// SIMATIC S7-200 project (STEP 7-Micro/WIN), CPU 226 REL 01.00

SYMBOL_TABLE SYM1
命令               VB100
bcc              VB101
bcc_ath          VB102
bcc_0            VB103
地址半高             VB104
地址半低             VB105
返回BCC            VB106
地址               VD110
位数h              VB114
位数               VB115
接收缓冲开始           VB120
接收缓冲结束           VB148
发送缓冲开始           VB149
发送缓冲结束           VB190
接受错缓冲开始          VB191
接受错缓冲结束          VB194
写到plc正确缓冲开始      VB195
写到plc正确缓冲结束      VB198
END_SYMBOL_TABLE

ORGANIZATION_BLOCK MAIN:OB1
TITLE=【101】环保处理厂的焚烧炉PLC控制程序
// 系统通过PLC管理焚烧炉的启动、运行、停止和故障处理，支持多设备协同工作。
// 操作员通过置位系统启动标志启动系统，随后系统根据1#燃烧室温度传感器和2#燃烧室温度传感器的反馈自动运行。焚烧过程由1#燃烧室燃烧器控制、2#燃烧室1#燃烧器控制和2#燃烧室2#燃烧器控制负责，但1#燃烧室燃烧器控制只能在2#燃烧室1#燃烧器控制未运行时启动，同样2#燃烧室1#燃烧器控制只能在1#燃烧室燃烧器控制未运行时启动，以防止焚烧炉过热或设备损坏。废液通过酸性废液输送泵控制和碱性废液输送泵控制输送，其中酸性废液输送泵控制和碱性废液输送泵控制交替运行，确保废液分开输送。接着，酸性废液喷嘴控制、碱性废液喷嘴控制和502废液喷嘴控制负责将废液喷射到焚烧炉内，且酸性废液喷嘴控制在废液输送时打开，确保废液均匀分布。
// 炉内气流由引风机控制和鼓风机控制维持，两者协同运行，保证氧气供应和废气排放顺畅。焚烧后的废渣由出渣机控制排出，且出渣机控制在焚烧结束后启动，避免堵塞。废气处理依赖药剂输送泵1控制至药剂输送泵4控制输送中和剂，其中药剂输送泵1控制在药剂可用时运行，防止泵空转；药剂池搅拌机控制确保药剂均匀。随后，能量回收通过余热锅炉1#给水泵控制和余热锅炉2#给水泵控制实现，余热锅炉1#给水泵控制在需要补水时启动，避免锅炉过压。
// 废气进一步通过喷淋塔电动阀控制和石灰池电磁阀控制处理，其中喷淋塔电动阀控制根据废气温度调整，确保处理效果。1#冷却塔风扇控制和2#冷却塔风扇控制冷却循环水，软水冷却泵控制辅助冷却。系统配备故障检测，如超温、熄火等，异常时通过故障报警灯控制提示操作员。停止时，系统启动标志复位，所有设备（如1#燃烧室燃烧器控制等）随之复位，确保安全关闭。
BEGIN
Network 1
LD     SM0.1
MOVB   16#9, SMB30           //口1波特率9600,N,8,1
ATCH   INT_0:INT0, 8         //口1中断,中断程序0
MOVW   16#3032, VW104        //PLC地址(01)0-30,1-31
MOVD   16#3030705, VD191     //VB191=3,VB192=3,7,5
R      M0.0, 8               //初始化MB0
MOVD   16#3030605, VD195     //接收错缓冲区
ENI
Network 2
LD     SM0.7
=      SM30.0
?000
Network 3
LD     M0.3                  //接收正确
O      M0.4                  //接收错
CALL   SBR_0:SBR0            //答复计算机
Network 4 // 子程序调用
// 
// 
LD     SM0.0
CALL   SBR_1:SBR1
CALL   SBR_2:SBR2
CALL   SBR_3:SBR3
CALL   SBR_4:SBR4
Network 5 // 系统启动
// 
// 
LD     M6.6
=      M10.0
Network 6
LD     SM0.0
MOVR   VD208, VD600
-R     5.0, VD600
MOVR   VD212, VD604
-R     5.0, VD604
MOVR   VD228, VD608
-R     5.0, VD608
MOVR   VD236, VD612
-R     5.0, VD612
MOVR   VD224, VD616
-R     5.0, VD616
MOVR   VD232, VD620
-R     5.0, VD620
Network 7 // 系统启动   1#燃烧室燃烧器控制
//  
// NETWORK COMMENTS
//  
// 
LD     SM0.0
A      M10.0
LPS
A      M6.5
LPS
S      Q4.1, 1
AR<    VD1216, VD600
S      Q4.2, 1
LRD
AR<    VD1216, VD604
S      Q4.3, 1
LRD
AR>    VD1216, VD208
R      Q4.2, 2
LRD
AR>    VD1216, VD212
R      Q4.3, 1
LPP
A      M14.1
R      Q4.2, 2
LPP
AN     M6.5
R      Q4.1, 3
Network 8 // 2#燃烧室1#燃烧器控制
//  
// NETWORK COMMENTS
//  
// 
LD     SM0.0
A      M10.0
LPS
A      M11.1
LPS
S      Q4.4, 1
AR<    VD1416, VD608
S      Q4.6, 1
LRD
AR<    VD1416, VD612
S      Q4.5, 1
LRD
AR>    VD1416, VD228
R      Q4.6, 1
LRD
AR>    VD1416, VD236
R      Q4.5, 1
LPP
A      M14.2
R      Q4.5, 2
LPP
AN     M11.1
R      Q4.4, 3
Network 9 // 2#燃烧室2#燃烧器控制
//  
// NETWORK COMMENTS
//  
// 
LD     SM0.0
A      M10.0
LPS
A      M11.3
LPS
S      Q4.7, 1
AR<    VD1416, VD616
S      Q5.1, 1
LRD
AR<    VD1416, VD620
S      Q5.0, 1
LRD
AR>    VD1416, VD224
R      Q5.1, 1
LRD
AR>    VD1416, VD232
R      Q5.0, 1
LPP
A      M14.3
R      Q5.0, 2
LPP
AN     M11.3
R      Q4.7, 3
Network 10 // 酸性废液输送泵控制
// 
// 
LD     SM0.0
LPS
A      M10.0
A      M10.2
S      Q2.3, 1
LPP
AN     M10.2
R      Q2.3, 1
Network 11 // 碱性废液输送泵控制
// 
// 
LD     SM0.0
LPS
A      M10.0
A      M10.4
S      Q2.4, 1
LPP
AN     M10.4
R      Q2.4, 1
Network 12 // 酸性废液喷嘴控制
// 
// 
LD     SM0.0
LPS
A      M10.0
A      M10.6
S      Q3.1, 1
LPP
AN     M10.6
R      Q3.1, 1
Network 13 // 碱性废液喷嘴控制
// 
// 
LD     SM0.0
LPS
A      M10.0
A      M1.0
S      Q3.2, 1
LPP
AN     M1.0
R      Q3.2, 1
Network 14 // 502废液喷嘴控制
// 
// 
LD     SM0.0
LPS
A      M10.0
A      M1.2
S      Q3.3, 1
LPP
AN     M1.2
R      Q3.3, 1
Network 15 // 引风机、鼓风机、风门执行器控制
// 
// 
LD     M10.0
LPS
A      M1.5
S      Q1.4, 1
LRD
A      Q1.4
A      M1.5
S      Q2.2, 1
LRD
AN     M1.4
R      Q2.2, 1
LPP
AN     M1.5
AN     Q2.2
R      Q1.4, 1
Network 16 // 出渣机控制
// 
// 
LD     SM0.0
A      M10.0
LPS
A      M1.6
S      Q1.2, 1
LPP
AN     M1.6
R      Q1.2, 1
Network 17 // 药剂输送泵、药剂池搅拌机控制
// 
// 
LD     SM0.0
LPS
A      M10.0
LPS
A      M2.1
S      Q1.5, 1
LRD
A      M2.3
S      Q1.6, 1
LRD
A      M2.5
S      Q1.7, 1
LRD
A      M2.7
S      Q2.0, 1
LPP
A      M3.1
S      Q2.1, 1
LPP
LPS
AN     M2.1
R      Q1.5, 1
LRD
AN     M2.3
R      Q1.6, 1
LRD
AN     M2.5
R      Q1.7, 1
LRD
AN     M2.7
R      Q2.0, 1
LPP
AN     M3.1
R      Q2.1, 1
Network 18 // 1#、2#给水泵控制
// 
// 
LD     SM0.0
LPS
A      M10.0
LPS
A      M3.3
S      Q0.2, 1
LPP
A      M3.5
S      Q0.3, 1
LPP
LPS
AN     M3.5
R      Q0.3, 1
LPP
AN     M3.3
R      Q0.2, 1
Network 19 // 502予处理罐蒸汽电磁阀、搅拌电机控制
// 
// 
LD     SM0.0
LPS
A      M10.0
LPS
AR<=   VD1116, VD204
S      Q3.5, 1
LPP
A      M3.7
S      Q0.6, 1
LPP
LPS
AN     M3.7
R      Q0.6, 1
LPP
AR>=   VD1116, VD200
R      Q3.5, 1
Network 20 // 余热锅炉给水泵控制
// 
// 
LD     SM0.0
LPS
A      M10.0
LPS
LD     M6.1
O      M16.2
ALD
AN     M16.1
S      Q0.4, 1
LRD
A      Q0.4
S      M16.0, 1
LRD
LD     M6.3
O      M16.2
ALD
AN     M16.0
S      Q0.5, 1
LPP
A      Q0.5
S      M16.1, 1
LPP
LPS
A      I0.0
AN     M16.3
=      M16.2
LRD
A      I0.3
AN     M16.3
R      Q0.4, 2
LRD
A      M6.2
R      Q0.4, 1
S      M16.3, 1
R      M16.0, 1
LRD
A      M6.4
R      Q0.5, 1
S      M16.3, 1
R      M16.1, 1
LPP
LD     M6.1
O      M6.3
ALD
R      M16.3, 1
Network 21 // 自吸泵控制
// 
// 
LD     SM0.0
LPS
A      M10.0
LPS
A      M4.1
S      Q2.5, 1
LRD
A      M4.3
S      Q2.6, 1
LPP
A      M4.5
S      Q2.7, 1
LPP
LPS
AN     M4.1
R      Q2.5, 1
LRD
AN     M4.3
R      Q2.6, 1
LPP
AN     M4.5
R      Q2.7, 1
Network 22 // 喷淋塔电动阀控制
// 
// 
LD     M10.0
MOVW   AIW12, AQW4
MOVW   AIW14, AQW12
S      Q3.6, 2
Network 23 // 软水冷却泵控制
// 
// 
LD     SM0.0
LPS
A      M10.0
A      M4.7
S      Q3.0, 1
LPP
AN     M4.7
R      Q3.0, 1
Network 24 // 上料提升机控制
// 
// 
LD     SM0.0
LPS
A      M10.0
LPS
A      M2.2
S      Q3.4, 1
LRD
AN     I1.0
R      Q3.4, 1
LRD
A      M5.2
S      Q5.5, 1
LPP
AN     I1.1
R      Q5.5, 1
LPP
A      M1.3
R      Q3.4, 1
R      Q5.5, 1
Network 25 // 冷却塔风扇电机
// 
// 
LD     SM0.0
LPS
A      M10.0
LPS
A      M5.3
S      Q0.0, 1
LPP
A      M5.5
S      Q0.1, 1
LPP
LPS
AN     M5.3
R      Q0.0, 1
LPP
AN     M5.5
R      Q0.1, 1
Network 26 // 石灰池电磁阀控制
LD     SM0.0
LPS
A      M10.0
LD     M5.7
O      I1.4
ALD
S      Q4.0, 1
R      M3.6, 1
LPP
LD     M6.0
O      I1.6
ALD
R      Q4.0, 1
S      M3.6, 1
Network 27 // 系统停止
LDN    M10.0
R      Q0.0, 1
R      Q0.1, 1
R      Q0.2, 1
R      Q0.3, 1
R      Q0.4, 1
R      Q0.5, 1
R      Q0.6, 1
R      Q0.7, 1
R      Q1.0, 1
R      Q1.1, 1
R      Q1.2, 1
R      Q1.3, 1
R      Q1.4, 1
R      Q1.5, 1
R      Q1.6, 1
R      Q1.7, 1
R      Q2.0, 1
R      Q2.1, 1
R      Q2.2, 1
R      Q2.3, 1
R      Q2.4, 1
R      Q2.5, 1
R      Q2.6, 1
R      Q2.7, 1
R      Q3.0, 1
R      Q3.1, 1
R      Q3.2, 1
R      Q3.3, 1
R      Q3.4, 1
R      Q3.5, 1
R      Q3.6, 1
Network 28 // 系统停止
LDN    M10.0
R      Q3.7, 1
R      Q4.0, 1
R      Q4.1, 1
R      Q4.2, 1
R      Q4.3, 1
R      Q4.4, 1
R      Q4.5, 1
R      Q4.6, 1
R      Q4.7, 1
R      Q5.0, 1
R      Q5.1, 1
R      Q5.4, 1
END_ORGANIZATION_BLOCK

SUBROUTINE_BLOCK SBR_0:SBR0
TITLE=
BEGIN
Network 2
LDB=   命令:VB100, 1           //读指令
A      M0.3                  //BCC正确
ATH    接收缓冲开始:VB120, VB110, 10
FILL   16#3030, VW152, 8     //将发送缓冲区清零
HTA    *地址:VD110, VB152, 位数h:VB114
MOVW   16#306, VW150         //置首标3,6
MOVB   5, VB170              //置结束符号,5
MOVB   21, 发送缓冲开始:VB149      //置发送字节数
Network 3 // 计算校验和
LDB=   命令:VB100, 1
A      M0.3
MOVD   &VB152, AC1           //指向发送缓冲区头
MOVB   0, 返回BCC:VB106        //初始化发送BCC
Network 4
LDB=   命令:VB100, 1
A      M0.3
FOR    AC0, +0, +15          //开始计算BCC
Network 5
LD     SM0.0
XORB   *AC1, 返回BCC:VB106
Network 6
LD     SM0.0
INCD   AC1
Network 7
NEXT
Network 8
LD     M0.3
AB=    命令:VB100, 1
HTA    返回BCC:VB106, VB168, 2 //将BCC HTA
XMT    发送缓冲开始:VB149, 0       //开始发送
R      M0.3, 1
Network 9
LDB=   命令:VB100, 2           //计算机写数据
A      M0.3                  //BCC正确
ATH    接收缓冲开始:VB120, VB110, 10 //分离出PLC区地址信息及字节数
ATH    VB130, *地址:VD110, 位数h:VB114 //将数据直接转换到直接地址
XMT    写到plc正确缓冲开始:VB195, 0  //返回给计算机3,6,5
R      M0.3, 1
Network 10
LD     M0.4                  //计算机来的数据BCC错返回给计算机3,7,5
XMT    接受错缓冲开始:VB191, 0
R      M0.4, 1
Network 11
//  RET
// 
END_SUBROUTINE_BLOCK

SUBROUTINE_BLOCK SBR_1:SBR1
TITLE=
BEGIN
Network 1 // 初始化
//  
// NETWORK COMMENTS
//  
// 
LD     SM0.1
MOVB   0, VB2600
MOVD   +0, VD1004
MOVD   +0, VD1104
MOVD   +0, VD1204
MOVD   +0, VD1304
MOVD   +0, VD1404
MOVD   +0, VD1504
MOVD   +0, VD1604
MOVD   +0, VD1704
MOVD   +0, VD1804
MOVD   +0, VD1904
MOVD   +0, VD2004
MOVD   +0, VD2104
MOVD   +0, VD2204
MOVD   +0, VD2304
MOVD   +0, VD2404
Network 2
LD     SM0.1
MOVD   +0, VD2504
MOVD   +0, VD1008
MOVD   +0, VD1108
MOVD   +0, VD1208
MOVD   +0, VD1308
MOVD   +0, VD1408
MOVD   +0, VD1508
MOVD   +0, VD1608
MOVD   +0, VD1708
MOVD   +0, VD1808
MOVD   +0, VD1908
MOVD   +0, VD2008
MOVD   +0, VD2108
MOVD   +0, VD2208
MOVD   +0, VD2308
MOVD   +0, VD2408
Network 3
LD     SM0.1
MOVD   +0, VD2508
MOVD   +0, VD1012
MOVD   +0, VD1112
MOVD   +0, VD1212
MOVD   +0, VD1312
MOVD   +0, VD1412
MOVD   +0, VD1512
MOVD   +0, VD1612
MOVD   +0, VD1712
MOVD   +0, VD1812
MOVD   +0, VD1912
MOVD   +0, VD2012
MOVD   +0, VD2112
MOVD   +0, VD2212
MOVD   +0, VD2312
MOVD   +0, VD2412
Network 4
LD     SM0.1
MOVD   +0, VD2512
R      Q0.0, 44
R      M16.0, 2
END_SUBROUTINE_BLOCK

SUBROUTINE_BLOCK SBR_2:SBR2
TITLE=
BEGIN
Network 1 // 软水箱温度 传感器故障
//  
// NETWORK COMMENTS
//  
// 
LD     SM0.0
LPS
LDR>=  VD1016, 205.9
OR<=   VD1016, 0.0
ALD
TON    T100, +100
LPP
A      T100
=      M12.0
Network 2 // 502予处理罐温度传感器故障
//  
// NETWORK COMMENTS
//  
// 
LD     SM0.0
LPS
LDR>=  VD1116, 205.9
OR<=   VD1116, 0.0
ALD
TON    T101, +100
LPP
A      T101
=      M12.1
Network 3 // 1#燃烧器温度传感器故障
LD     SM0.0
LPS
LDR>=  VD1216, 1132.0
OR<=   VD1216, 0.0
ALD
TON    T102, +100
LPP
A      T102
=      M12.2
Network 4 // 炉膛负压传感器故障
LD     SM0.0
LPS
LDR>=  VD1316, 200.0
OR<=   VD1316, 0.0
ALD
TON    T103, +100
LPP
A      T103
=      M12.3
Network 5 // 2#燃烧室2#燃烧器温度传感器故障
LD     SM0.0
LPS
LDR>=  VD1416, 1338.0
OR<=   VD1416, 0.0
ALD
TON    T104, +100
LPP
A      T104
=      M12.4
Network 6 // 锅炉出口温度传感器故障
LD     SM0.0
LPS
LDR>=  VD1516, 823.0
OR<=   VD1516, 0.0
ALD
TON    T105, +100
LPP
A      T105
=      M12.5
Network 7 // 1#喷淋塔出口温度传感器故障
LD     SM0.0
LPS
LDR>=  VD1616, 411.8
OR<=   VD1616, 0.0
ALD
TON    T106, +100
LPP
A      T106
=      M12.6
Network 8 // 2#喷淋塔出口温度传感器故障
LD     SM0.0
LPS
LDR>=  VD1716, 308.9
OR<=   VD1716, 0.0
ALD
TON    T107, +100
LPP
A      T107
=      M12.7
Network 9 // 2#喷淋塔水温温度传感器故障
LD     SM0.0
LPS
LDR>=  VD1816, 205.9
OR<=   VD1816, 0.0
ALD
TON    T108, +100
LPP
A      T108
=      M13.0
Network 10 // 喷淋塔水池温度传感器故障
LD     SM0.0
LPS
LDR>=  VD1916, 205.9
OR<=   VD1916, 0.0
ALD
TON    T109, +100
LPP
A      T109
=      M13.1
Network 11 // 引风机反馈故障
LD     SM0.0
LPS
LDR>=  VD2316, 90.0
OR<=   VD2316, 0.0
ALD
TON    T111, +100
LPP
A      T111
=      M13.3
Network 12 // 鼓风机反馈故障
LD     SM0.0
LPS
LDR>=  VD2416, 90.0
OR<=   VD2416, 0.0
ALD
TON    T112, +100
LPP
A      T112
=      M13.4
Network 13 // 工作油位计故障
LD     SM0.0
LPS
LDR>=  VD2516, 1500.0
OR<=   VD2516, 0.0
ALD
TON    T113, +100
LPP
A      T113
=      M13.5
Network 14 // 1#燃烧室超温故障
LD     SM0.0
MOVD   VD208, VD260
+D     +200, VD260
AR>=   VD1216, VD260
=      M13.6
Network 15 // 2#燃烧室超温故障
LD     SM0.0
MOVD   VD236, VD264
+D     +100, VD264
AR>=   VD1416, VD264
=      M13.7
Network 16 // 1#燃烧器熄火故障
LD     I0.4
=      M14.1
Network 17 // 2#燃烧室1#燃烧器熄火故障
LD     I0.7
=      M14.2
Network 18 // 2#燃烧室2#燃烧器熄火故障
LD     I1.2
=      M14.3
Network 19 // 余热锅炉水位极低
LD     I0.2
=      M14.4
Network 20 // 工作油位极低故障
LDR<=  VD2516, VD240
=      M14.6
Network 21 // 沉淀池液位极低
LDN    I1.3
=      M14.7
Network 22 // 沉淀池液位极高
LDN    I1.7
=      M15.0
Network 23 // 余热锅炉压力过高
LDN    I0.6
=      M15.3
Network 24 // 故障报警
// 
// 
LD     M12.0
O      M12.1
O      M12.2
O      M12.3
O      M12.4
O      M12.5
O      M12.6
O      M12.7
O      M13.0
O      M13.1
O      M13.3
O      M13.4
O      M13.5
O      M13.6
O      M13.7
O      M14.1
O      M14.2
O      M14.3
O      M14.4
O      M14.6
O      M14.7
O      M15.0
O      M15.1
S      M2.4, 1
Network 25 // 故障消除
LD     SM0.0
LPS
A      M2.4
LPS
AN     T115
TON    T114, +100
LPP
AN     M15.5
AN     M15.2
=      M16.4
LRD
LPS
A      T114
S      M15.5, 1
LRD
A      M15.5
TON    T115, +40
LPP
A      T115
R      M15.5, 1
LPP
A      I1.5
R      M2.4, 1
R      M15.2, 1
Network 26 // 消音
// 
// 
LD     M1.1
S      M15.2, 1
Network 27
LD     M16.4
=      Q5.6
END_SUBROUTINE_BLOCK

SUBROUTINE_BLOCK SBR_3:SBR3
TITLE=
BEGIN
Network 1 // 模拟量处理
//  
// NETWORK COMMENTS
//  
// 
LD     SM0.0
MOVW   AIW0, VW1002
MOVW   AIW2, VW1102
MOVW   AIW4, VW1202
MOVW   AIW6, VW1302
MOVW   AIW8, VW1402
MOVW   AIW10, VW1502
MOVW   AIW12, VW1602
MOVW   AIW14, VW1702
MOVW   AIW16, VW1802
MOVW   AIW18, VW1902
MOVW   AIW20, VW2002
MOVW   AIW22, VW2102
MOVW   AIW24, VW2202
MOVW   AIW26, VW2302
MOVW   AIW28, VW2402
MOVW   AIW30, VW2502
Network 2
LDW>=  VW1002, +0
MOVW   +0, VW1000
NOT
MOVW   16#FFFF, VW1000
Network 3
LDW>=  VW1102, +0
MOVW   +0, VW1100
NOT
MOVW   16#FFFF, VW1100
Network 4
LDW>=  VW1202, +0
MOVW   +0, VW1200
NOT
MOVW   16#FFFF, VW1200
Network 5
LDW>=  VW1302, +0
MOVW   +0, VW1300
NOT
MOVW   16#FFFF, VW1300
Network 6
LDW>=  VW1402, +0
MOVW   +0, VW1400
NOT
MOVW   16#FFFF, VW1400
Network 7
LDW>=  VW1502, +0
MOVW   +0, VW1500
NOT
MOVW   16#FFFF, VW1500
Network 8
LDW>=  VW1602, +0
MOVW   +0, VW1600
NOT
MOVW   16#FFFF, VW1600
Network 9
LDW>=  VW1702, +0
MOVW   +0, VW1700
NOT
MOVW   16#FFFF, VW1700
Network 10
LDW>=  VW1802, +0
MOVW   +0, VW1800
NOT
MOVW   16#FFFF, VW1800
Network 11
LDW>=  VW1902, +0
MOVW   +0, VW1900
NOT
MOVW   16#FFFF, VW1900
Network 12
LDW>=  VW2002, +0
MOVW   +0, VW2000
NOT
MOVW   16#FFFF, VW2000
Network 13
LDW>=  VW2102, +0
MOVW   +0, VW2100
NOT
MOVW   16#FFFF, VW2100
Network 14
LDW>=  VW2202, +0
MOVW   +0, VW2200
NOT
MOVW   16#FFFF, VW2200
Network 15
LDW>=  VW2302, +0
MOVW   +0, VW2300
NOT
MOVW   16#FFFF, VW2300
Network 16
LDW>=  VW2402, +0
MOVW   +0, VW2400
NOT
MOVW   16#FFFF, VW2400
Network 17
LDW>=  VW2502, +0
MOVW   +0, VW2500
NOT
MOVW   16#FFFF, VW2500
Network 18 // 求和
// 
// 
LD     SM0.0
+D     VD1000, VD1004
+D     VD1100, VD1104
+D     VD1200, VD1204
+D     VD1300, VD1304
+D     VD1400, VD1404
+D     VD1500, VD1504
+D     VD1600, VD1604
+D     VD1700, VD1704
+D     VD1800, VD1804
+D     VD1900, VD1904
+D     VD2000, VD2004
+D     VD2100, VD2104
+D     VD2200, VD2204
+D     VD2300, VD2304
+D     VD2400, VD2404
+D     VD2500, VD2504
Network 19
LD     SM0.0
INCB   VB2600
Network 20
LDB>=  VB2600, 16
MOVD   VD1004, VD1008
MOVD   VD1104, VD1108
MOVD   VD1204, VD1208
MOVD   VD1304, VD1308
MOVD   VD1404, VD1408
MOVD   VD1504, VD1508
MOVD   VD1604, VD1608
MOVD   VD1704, VD1708
MOVD   VD1804, VD1808
MOVD   VD1904, VD1908
MOVD   VD2004, VD2008
MOVD   VD2104, VD2108
MOVD   VD2204, VD2208
MOVD   VD2304, VD2308
MOVD   VD2404, VD2408
MOVD   VD2504, VD2508
Network 21
LDB>=  VB2600, 16
MOVD   +0, VD1004
MOVD   +0, VD1104
MOVD   +0, VD1204
MOVD   +0, VD1304
MOVD   +0, VD1404
MOVD   +0, VD1504
MOVD   +0, VD1604
MOVD   +0, VD1704
MOVD   +0, VD1804
MOVD   +0, VD1904
MOVD   +0, VD2004
MOVD   +0, VD2104
MOVD   +0, VD2204
MOVD   +0, VD2304
MOVD   +0, VD2404
Network 22 // 平均值
// 
// 
LDB>=  VB2600, 16
MOVD   +0, VD2504
SRD    VD1008, 4
SRD    VD1108, 4
SRD    VD1208, 4
SRD    VD1308, 4
SRD    VD1408, 4
SRD    VD1508, 4
SRD    VD1608, 4
SRD    VD1708, 4
SRD    VD1808, 4
SRD    VD1908, 4
SRD    VD2008, 4
SRD    VD2108, 4
SRD    VD2208, 4
SRD    VD2308, 4
SRD    VD2408, 4
Network 23
LDB>=  VB2600, 16
SRD    VD2508, 4
MOVB   0, VB2600
Network 24
LD     SM0.0
MOVD   VD1008, VD1024
MOVD   VD1108, VD1124
MOVD   VD1208, VD1224
MOVD   VD1308, VD1324
MOVD   VD1408, VD1424
MOVD   VD1508, VD1524
MOVD   VD1608, VD1624
MOVD   VD1708, VD1724
MOVD   VD1808, VD1824
MOVD   VD1908, VD1924
MOVD   VD2008, VD2024
MOVD   VD2108, VD2124
MOVD   VD2208, VD2224
MOVD   VD2308, VD2324
MOVD   VD2408, VD2424
MOVD   VD2508, VD2524
Network 25
LD     SM0.0
DTR    VD1024, VD1024
DTR    VD1124, VD1124
DTR    VD1224, VD1224
DTR    VD1324, VD1324
DTR    VD1424, VD1424
DTR    VD1524, VD1524
DTR    VD1624, VD1624
DTR    VD1724, VD1724
DTR    VD1824, VD1824
DTR    VD1924, VD1924
DTR    VD2024, VD2024
DTR    VD2124, VD2124
DTR    VD2224, VD2224
DTR    VD2324, VD2324
DTR    VD2424, VD2424
DTR    VD2524, VD2524
Network 26
LD     SM0.0
MOVR   VD1024, VD1012
MOVR   VD1124, VD1112
MOVR   VD1224, VD1212
MOVR   VD1324, VD1312
MOVR   VD1424, VD1412
MOVR   VD1524, VD1512
MOVR   VD1624, VD1612
MOVR   VD1724, VD1712
MOVR   VD1824, VD1812
MOVR   VD1924, VD1912
MOVR   VD2024, VD2012
MOVR   VD2124, VD2112
MOVR   VD2224, VD2212
MOVR   VD2324, VD2312
MOVR   VD2424, VD2412
MOVR   VD2524, VD2512
Network 27
LD     SM0.0
-R     6400.0, VD1012
-R     6400.0, VD1112
-R     6400.0, VD1212
-R     6400.0, VD1312
-R     6400.0, VD1412
-R     6400.0, VD1512
-R     6400.0, VD1612
-R     6400.0, VD1712
-R     6400.0, VD1812
-R     6400.0, VD1912
-R     6400.0, VD2012
-R     6400.0, VD2112
-R     6400.0, VD2212
-R     0.0, VD2312
-R     0.0, VD2412
-R     6400.0, VD2512
Network 28
LD     SM0.0
/R     25600.0, VD1012
/R     25600.0, VD1112
/R     25600.0, VD1212
/R     25600.0, VD1312
/R     22400.0, VD1412
/R     25600.0, VD1512
/R     25600.0, VD1612
/R     25600.0, VD1712
/R     25600.0, VD1812
/R     25600.0, VD1912
/R     25600.0, VD2012
/R     25600.0, VD2112
/R     25600.0, VD2212
/R     16000.0, VD2312
/R     16000.0, VD2412
/R     25600.0, VD2512
Network 29
LD     SM0.0
*R     200.0, VD1012
*R     200.0, VD1112
*R     1100.0, VD1212
*R     200.0, VD1312
*R     1300.0, VD1412
*R     800.0, VD1512
*R     400.0, VD1612
*R     300.0, VD1712
*R     200.0, VD1812
*R     200.0, VD1912
*R     100.0, VD2012
*R     100.0, VD2112
*R     100.0, VD2212
*R     99.0, VD2312
*R     127.0, VD2412
*R     100.0, VD2512
Network 30
LD     SM0.0
-R     11.3, VD2412
-R     7.0, VD2312
+R     6.5, VD1312
Network 31
LD     SM0.0
-R     90.0, VD2412
*R     -1.0, VD2412
-R     30.0, VD1312
+R     0.0, VD1412
Network 32
LD     SM0.0
MOVR   VD1012, VD1016
MOVR   VD1112, VD1116
MOVR   VD1212, VD1216
MOVR   VD1312, VD1316
MOVR   VD1412, VD1416
MOVR   VD1512, VD1516
MOVR   VD1612, VD1616
MOVR   VD1712, VD1716
MOVR   VD1812, VD1816
MOVR   VD1912, VD1916
MOVR   VD2012, VD2016
MOVR   VD2112, VD2116
MOVR   VD2212, VD2216
MOVR   VD2312, VD2316
MOVR   VD2412, VD2416
MOVR   VD2512, VD2516
END_SUBROUTINE_BLOCK

SUBROUTINE_BLOCK SBR_4:SBR4
TITLE=MCGS模拟量处理模块 
// 
BEGIN
Network 1 // PLC-MCGS数据处理（保留一位小数点）   软水箱温度处理
// 
// 
LD     SM0.0
MOVR   VD1016, VD1020
*R     10.0, VD1020
TRUNC  VD1020, VD1020
MOVW   VW1022, VW300
Network 2 // 502予处理罐温度处理
LD     SM0.0
MOVR   VD1116, VD1120
*R     10.0, VD1120
TRUNC  VD1120, VD1120
MOVW   VW1122, VW302
Network 3 // 燃烧室1温度处理
// 
// 
LD     SM0.0
MOVR   VD1216, VD1220
*R     10.0, VD1220
TRUNC  VD1220, VD1220
MOVW   VW1222, VW304
Network 4 // 炉膛负压处理
LD     SM0.0
MOVR   VD1316, VD1320
*R     10.0, VD1320
TRUNC  VD1320, VD1320
MOVW   VW1322, VW306
Network 5 // 燃烧室2温度处理
// 
// 
LD     SM0.0
MOVR   VD1416, VD1420
*R     10.0, VD1420
TRUNC  VD1420, VD1420
MOVW   VW1422, VW308
Network 6 // 锅炉出口烟道温度处理
// 
// 
LD     SM0.0
MOVR   VD1516, VD1520
*R     10.0, VD1520
TRUNC  VD1520, VD1520
MOVW   VW1522, VW310
Network 7 // 喷淋塔2出口烟道温度处理
// 
// 
LD     SM0.0
MOVR   VD1616, VD1620
*R     10.0, VD1620
TRUNC  VD1620, VD1620
MOVW   VW1622, VW312
Network 8 // 喷淋塔2出口烟道温度处理
// 
// 
LD     SM0.0
MOVR   VD1716, VD1720
*R     10.0, VD1720
TRUNC  VD1720, VD1720
MOVW   VW1722, VW314
Network 9 // 喷淋塔2水温度处理
// 
// 
LD     SM0.0
MOVR   VD1816, VD1820
*R     10.0, VD1820
TRUNC  VD1820, VD1820
MOVW   VW1822, VW316
Network 10 // 喷淋塔2水池温度处理
// 
// 
LD     SM0.0
MOVR   VD1916, VD1920
*R     10.0, VD1920
TRUNC  VD1920, VD1920
MOVW   VW1922, VW318
Network 11 // 余热锅炉压力处理
// 
// 
LD     SM0.0
MOVR   VD2216, VD2220
*R     10.0, VD2220
TRUNC  VD2220, VD2220
MOVW   VW2222, VW320
Network 12 // 引风机反馈信号处理
// 
// 
LD     SM0.0
MOVR   VD2316, VD2320
*R     10.0, VD2320
TRUNC  VD2320, VD2320
MOVW   VW2322, VW322
Network 13 // 鼓风机反馈信号处理
// 
// 
LD     SM0.0
MOVR   VD2416, VD2420
*R     10.0, VD2420
TRUNC  VD2420, VD2420
MOVW   VW2422, VW324
Network 14 // 工作油箱信号处理
// 
// 
LD     SM0.0
MOVR   VD2516, VD2520
*R     10.0, VD2520
TRUNC  VD2520, VD2520
MOVW   VW2522, VW326
Network 15 // MCGS-PLC数据处理   502予处理罐温度上限、下限设置处理
LD     SM0.0
MOVW   VW350, VW402
MOVW   VW352, VW406
MOVW   +0, VW400
MOVW   +0, VW404
DTR    VD400, VD400
DTR    VD404, VD404
MOVR   VD400, VD200
MOVR   VD404, VD204
Network 16 // 1#燃烧室温度上限、下限设置处理
LD     SM0.0
MOVW   VW354, VW410
MOVW   VW356, VW414
MOVW   +0, VW408
MOVW   +0, VW412
DTR    VD408, VD408
DTR    VD412, VD412
MOVR   VD408, VD208
MOVR   VD412, VD212
Network 17 // 炉膛负压上限、下限设置处理
// 
// 
LD     SM0.0
MOVW   VW358, VW418
MOVW   VW360, VW422
MOVW   +0, VW416
MOVW   +0, VW420
DTR    VD416, VD416
DTR    VD420, VD420
MOVR   VD416, VD216
MOVR   VD420, VD220
Network 18 // 2#燃烧室温度上限、下限设置处理
// 
// 
LD     SM0.0
MOVW   VW362, VW426
MOVW   VW364, VW430
MOVW   +0, VW424
MOVW   +0, VW428
DTR    VD424, VD424
DTR    VD428, VD428
MOVR   VD424, VD224
MOVR   VD428, VD228
Network 19 // 余热锅炉出口烟温上限设置处理
LD     SM0.0
MOVW   VW366, VW434
MOVW   +0, VW432
DTR    VD432, VD432
MOVR   VD432, VD232
MOVW   VW380, VW462
MOVW   +0, VW460
DTR    VD460, VD460
MOVR   VD460, VD260
Network 20 // 1#喷淋塔出口烟温上限设置处理
// 
// 
LD     SM0.0
MOVW   VW368, VW438
MOVW   +0, VW436
DTR    VD436, VD436
MOVR   VD436, VD236
Network 21 // 2#喷淋塔出口烟温上限设置处理
// 
// 
LD     SM0.0
MOVW   VW370, VW442
MOVW   +0, VW440
DTR    VD440, VD440
MOVR   VD440, VD240
Network 22 // 余热锅炉压力上限、下限设置处理
LD     SM0.0
MOVW   VW372, VW446
MOVW   VW374, VW450
MOVW   +0, VW444
MOVW   +0, VW448
DTR    VD444, VD444
DTR    VD448, VD448
MOVR   VD444, VD244
MOVR   VD448, VD248
Network 23 // 工作油位上限、下限设置处理
LD     SM0.0
MOVW   VW376, VW454
MOVW   VW378, VW458
MOVW   +0, VW452
MOVW   +0, VW456
DTR    VD452, VD452
DTR    VD456, VD456
MOVR   VD452, VD252
MOVR   VD456, VD256
END_SUBROUTINE_BLOCK

INTERRUPT_BLOCK INT_0:INT0
TITLE=
BEGIN
Network 2
LDB=   SMB2, 1               //首字节为命令位1表示读
OB=    SMB2, 2               //首字节为命令位1表示写
S      M0.0, 1               //收到首字节标志
R      M0.1, 7
MOVB   SMB2, 命令:VB100        //命令保存在VB100
MOVD   &接收缓冲开始:VB120, VD180  //VB120 为接收缓冲区开始
MOVB   0, bcc:VB101          //初始化BCC
Network 3
LD     M0.0
AB=    SMB2, 地址半高:VB104      //核对PLC站号H
S      M0.1, 1               //站号H核对通过
R      M0.0, 1
Network 4
LDB=   SMB2, 5               //是结束符吗
DECD   VD180                 //当发现结束符号的时候VB101中已经包括BCC本身
XORB   *VD180, bcc:VB101     //所以将BCC再次计算即可还原出不含BCC的BCC
DECD   VD180
XORB   *VD180, bcc:VB101
ATH    *VD180, bcc_ath:VB102, 2 //指针回到BCC处,还原出计算机的BCC
MOVB   bcc_ath:VB102, bcc_0:VB103 //判断计算的BCC和计算机的BCC是否相等
XORB   bcc:VB101, bcc_0:VB103
R      M0.2, 1
Network 5
LD     M0.2                  //如果已经收到PLC站号L则说明已经开始收数据
MOVB   SMB2, *VD180
INCD   VD180                 //指针+1
XORB   SMB2, bcc:VB101       //计算校验和
Network 6
LD     M0.1
AB=    SMB2, 地址半低:VB105      //核对PLC站号L
S      M0.2, 1               //置站号L正确标志
R      M0.1, 1
Network 7
LDB=   SMB2, 5               //判断结束符号
AB=    bcc_0:VB103, 0        //判断BCC
S      M0.3, 1               //如果BCC通过则置位M0.3�3
Network 8
LDB=   SMB2, 5               //判断结束符号
AB>=   bcc_0:VB103, 1        //判断BCC
S      M0.4, 1               //如果BCC未通过则置位M0.3�3
Network 9
//  RETI
// 
END_INTERRUPT_BLOCK
